FUNCTION_BLOCK AssemblyActuatorHorizontal EXTENDS ZEquipment.ActuatorDigitalBiLsPlusMinus

METHOD PUBLIC AtAssembly : BOOL
VAR_INPUT
END_VAR
AtAssembly := IsAtMinus();
END_METHOD

METHOD PUBLIC AtTransport : BOOL
VAR_INPUT
END_VAR
AtTransport := IsAtPlus();
END_METHOD

METHOD PUBLIC ToAssemblyAsync
VAR_INPUT
  startToken : ZCore.IStartToken;
END_VAR
MoveMinusAsync(startToken:=startToken);
END_METHOD

METHOD PUBLIC ToTransportAsync
VAR_INPUT
  startToken : ZCore.IStartToken;
END_VAR
MovePlusAsync(startToken:=startToken);
END_METHOD

END_FUNCTION_BLOCK

(* stored: Version 1.1.0.1
   POU AssemblyActuatorHorizontal: Id {5a6b0ae2-2644-488a-9e94-a94a5a3e6f46}, SpecialFunc None
   Method AtAssembly: Id {800cf822-9882-4b7f-b25d-ebc7e3302dc8}
   Method AtTransport: Id {6ab11686-3147-4a05-b4ab-0da8ea2c2a8f}
   Method ToAssemblyAsync: Id {e521c05d-d0ae-46d9-992d-05e16a1bb6c3}
   Method ToTransportAsync: Id {ca110a1f-47ed-421f-8b27-693236ec321d} *)
